{attribute 'GeneratedUsingTerminal: EL3783-0000-0018'}
{attribute addProperty BoxType "EL3783-0000-0018"}
{attribute addProperty Id "U1_SamplesAT %I*U1_Samples_1109DCAA40"}
{attribute addProperty CRC "2819058525"}
{attribute addProperty Size "40"}
TYPE L1_Voltage_Samples_A8076B5D :
STRUCT
	{attribute addProperty Name "U1_Samples"}
	U1_Samples AT %I* : U1_Samples_1109DCAA;
END_STRUCT
END_TYPE

(* stored: Version 1.2.0.0, ProductVersion 3.1.4024.9
   DUT L1_Voltage_Samples_A8076B5D: Id {43446ed8-6a94-4533-b751-4cfe94921804} *)
